FUNCTION_BLOCK ILOCK_BLOCK_A2X (* Prioritizes the first active input (Adapter Version, UP/DOWN fed from a single A2X input/output). *)
  (* Standard: 61499-2; Description: Copyright (c) 2026 HR Agrartechnik GmbH This program and the accompanying materials are made available under the terms of the Eclipse Public License 2.0 which is available at https://www.eclipse.org/legal/epl-2.0/ SPDX-License-Identifier: EPL-2.0 *)
  (* Version 1.0, 2026-09-05, Franz Höpfinger, HR Agrartechnik GmbH, initial API and implementation and/or initial documentation *)
  PACKAGE logiBUS::signalprocessing::interlock;
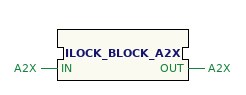
  SOCKETS
    IN : adapter::types::unidirectional::A2X; (* Input for forward/up and backward/down direction *)
  END_SOCKETS
  PLUGS
    OUT : adapter::types::unidirectional::A2X; (* Output for forward/up and backward/down direction *)
  END_PLUGS
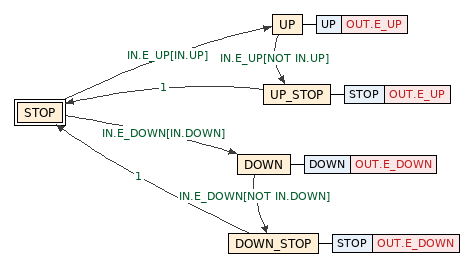
  EC_STATES
    STOP;
    UP : UP -> OUT.E_UP;
    DOWN : DOWN -> OUT.E_DOWN;
    UP_STOP : STOP -> OUT.E_UP;
    DOWN_STOP : STOP -> OUT.E_DOWN;
  END_STATES
  EC_TRANSITIONS
    STOP TO DOWN := IN.E_DOWN[IN.DOWN];
    STOP TO UP := IN.E_UP[IN.UP];
    DOWN TO DOWN_STOP := IN.E_DOWN[NOT IN.DOWN];
    UP TO UP_STOP := IN.E_UP[NOT IN.UP];
    DOWN_STOP TO STOP := 1;
    UP_STOP TO STOP := 1;
  END_TRANSITIONS
  ALGORITHM UP IN ST:
OUT.UP := BOOL#TRUE;
OUT.DOWN := BOOL#FALSE;
  END_ALGORITHM
  ALGORITHM DOWN IN ST:
OUT.UP := BOOL#FALSE;
OUT.DOWN := BOOL#TRUE;
  END_ALGORITHM
  ALGORITHM STOP IN ST:
OUT.UP := BOOL#FALSE;
OUT.DOWN := BOOL#FALSE;
  END_ALGORITHM
END_FUNCTION_BLOCK
